FUNCTION F_TB_Rx_BCC : BOOL
VAR_INPUT
	rxStr: STRING;
END_VAR
VAR
	i, len1, len2: INT;
	bArr: ARRAY[0..255] OF BYTE;
	b1: BYTE;
END_VAR

// SMC HEBC002-WA10
len1 := LEN(STR:=rxStr);
len2 := len1;
len1 := len1 - 1;
bArr := MAXSTRING_TO_BYTEARR(rxStr);
FOR i := 0 TO len1 DO
	b1 := b1 XOR bArr[i];
END_FOR
F_TB_Rx_BCC := b1 = bArr[len2];

END_FUNCTION

(* stored: Version 1.1.0.1, ProductVersion 3.1.4024.12
   POU F_TB_Rx_BCC: Id {6909b4a3-6bb0-43c2-bc3d-5c7c8ddd649d}, SpecialFunc None *)
